PROGRAM P5_02_DiagramVisualisation
VAR
END_VAR
VAR // added by the converter: edge detectors and wires of the graphical bodies
    _w1, _w2, _w3 : BOOL;
    _w4 : INT;
END_VAR

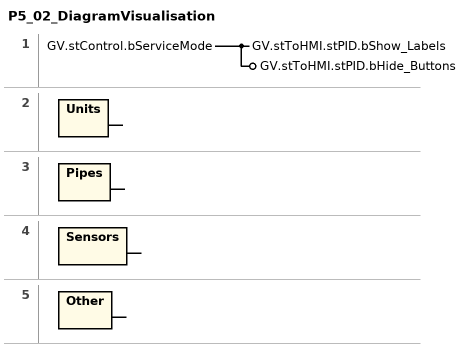
// NETWORK 1
_w1 := GV.stControl.bServiceMode;
GV.stToHMI.stPID.bShow_Labels := _w1;
GV.stToHMI.stPID.bHide_Buttons := NOT _w1;

// NETWORK 2
Units();

// NETWORK 3
Pipes();

// NETWORK 4
Sensors();

// NETWORK 5
Other();

ACTION Other:
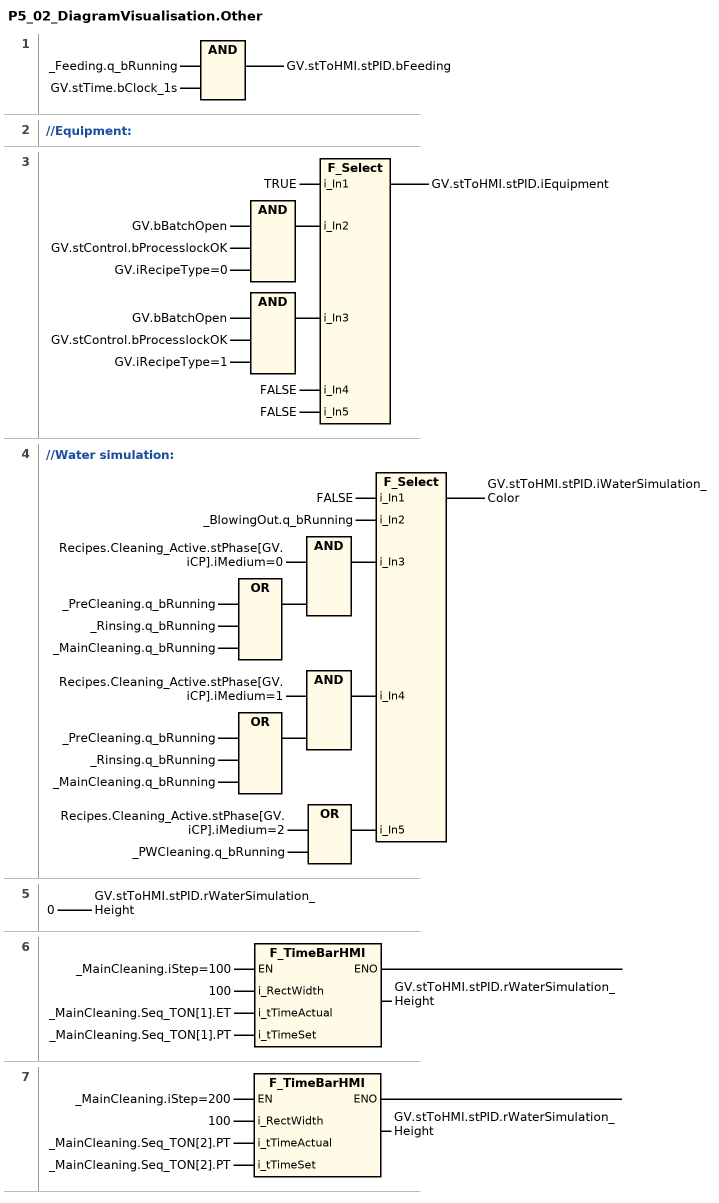
// NETWORK 1
GV.stToHMI.stPID.bFeeding := _Feeding.q_bRunning AND GV.stTime.bClock_1s;

// NETWORK 2
// label: //Equipment

// NETWORK 3
GV.stToHMI.stPID.iEquipment := F_Select(i_In1 := TRUE, i_In2 := GV.bBatchOpen AND GV.stControl.bProcesslockOK AND (GV.iRecipeType=0), i_In3 := GV.bBatchOpen AND GV.stControl.bProcesslockOK AND (GV.iRecipeType=1), i_In4 := FALSE, i_In5 := FALSE);

// NETWORK 4
// label: //Water simulation
GV.stToHMI.stPID.iWaterSimulation_Color := F_Select(i_In1 := FALSE, i_In2 := _BlowingOut.q_bRunning, i_In3 := (Recipes.Cleaning_Active.stPhase[GV.iCP].iMedium=0) AND (_PreCleaning.q_bRunning OR _Rinsing.q_bRunning OR _MainCleaning.q_bRunning), i_In4 := (Recipes.Cleaning_Active.stPhase[GV.iCP].iMedium=1) AND (_PreCleaning.q_bRunning OR _Rinsing.q_bRunning OR _MainCleaning.q_bRunning), i_In5 := (Recipes.Cleaning_Active.stPhase[GV.iCP].iMedium=2) OR _PWCleaning.q_bRunning);

// NETWORK 5
GV.stToHMI.stPID.rWaterSimulation_Height := 0;

// NETWORK 6
IF _MainCleaning.iStep=100 THEN
    GV.stToHMI.stPID.rWaterSimulation_Height := F_TimeBarHMI(i_RectWidth := 100, i_tTimeActual := _MainCleaning.Seq_TON[1].ET, i_tTimeSet := _MainCleaning.Seq_TON[1].PT);
END_IF

// NETWORK 7
IF _MainCleaning.iStep=200 THEN
    GV.stToHMI.stPID.rWaterSimulation_Height := F_TimeBarHMI(i_RectWidth := 100, i_tTimeActual := _MainCleaning.Seq_TON[2].PT, i_tTimeSet := _MainCleaning.Seq_TON[2].PT);
END_IF

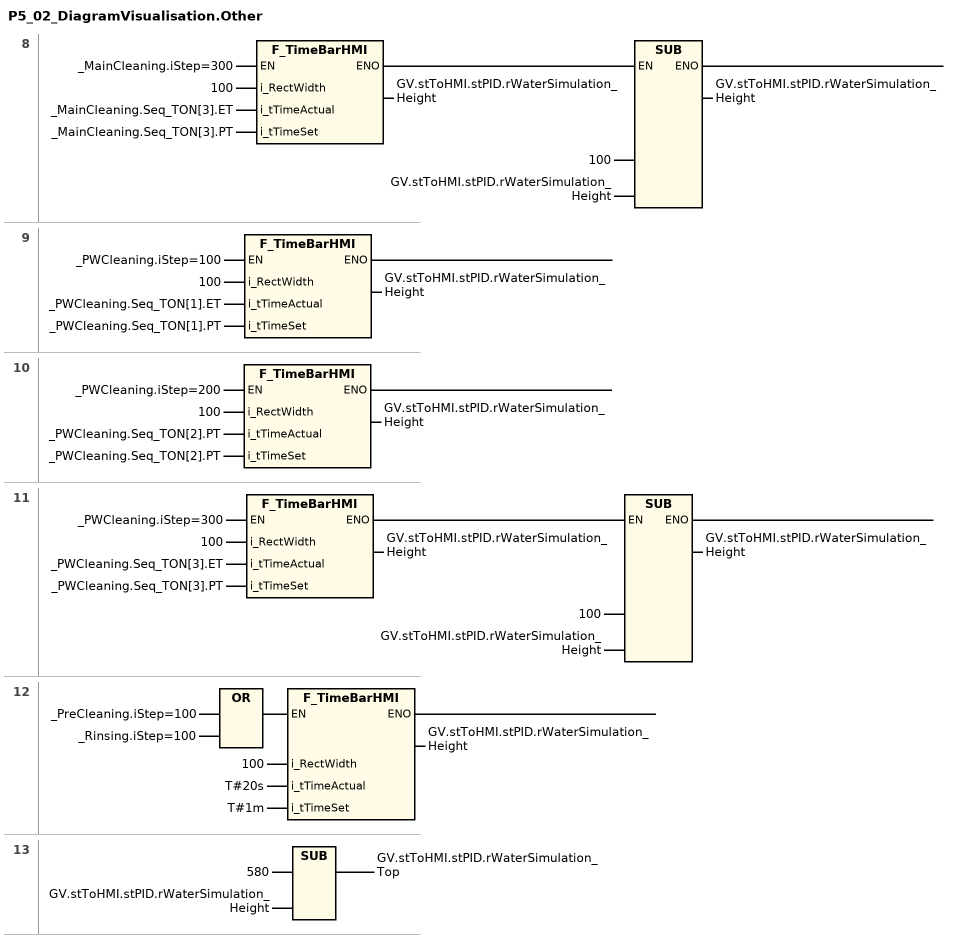
// NETWORK 8
_w2 := _MainCleaning.iStep=300;
IF _w2 THEN
    GV.stToHMI.stPID.rWaterSimulation_Height := F_TimeBarHMI(i_RectWidth := 100, i_tTimeActual := _MainCleaning.Seq_TON[3].ET, i_tTimeSet := _MainCleaning.Seq_TON[3].PT);
END_IF
IF _w2 THEN GV.stToHMI.stPID.rWaterSimulation_Height := 100 - GV.stToHMI.stPID.rWaterSimulation_Height; END_IF

// NETWORK 9
IF _PWCleaning.iStep=100 THEN
    GV.stToHMI.stPID.rWaterSimulation_Height := F_TimeBarHMI(i_RectWidth := 100, i_tTimeActual := _PWCleaning.Seq_TON[1].ET, i_tTimeSet := _PWCleaning.Seq_TON[1].PT);
END_IF

// NETWORK 10
IF _PWCleaning.iStep=200 THEN
    GV.stToHMI.stPID.rWaterSimulation_Height := F_TimeBarHMI(i_RectWidth := 100, i_tTimeActual := _PWCleaning.Seq_TON[2].PT, i_tTimeSet := _PWCleaning.Seq_TON[2].PT);
END_IF

// NETWORK 11
_w3 := _PWCleaning.iStep=300;
IF _w3 THEN
    GV.stToHMI.stPID.rWaterSimulation_Height := F_TimeBarHMI(i_RectWidth := 100, i_tTimeActual := _PWCleaning.Seq_TON[3].ET, i_tTimeSet := _PWCleaning.Seq_TON[3].PT);
END_IF
IF _w3 THEN GV.stToHMI.stPID.rWaterSimulation_Height := 100 - GV.stToHMI.stPID.rWaterSimulation_Height; END_IF

// NETWORK 12
IF (_PreCleaning.iStep=100) OR (_Rinsing.iStep=100) THEN
    GV.stToHMI.stPID.rWaterSimulation_Height := F_TimeBarHMI(i_RectWidth := 100, i_tTimeActual := T#20s, i_tTimeSet := T#1m);
END_IF

// NETWORK 13
GV.stToHMI.stPID.rWaterSimulation_Top := 580 - GV.stToHMI.stPID.rWaterSimulation_Height;
END_ACTION

ACTION Pipes:
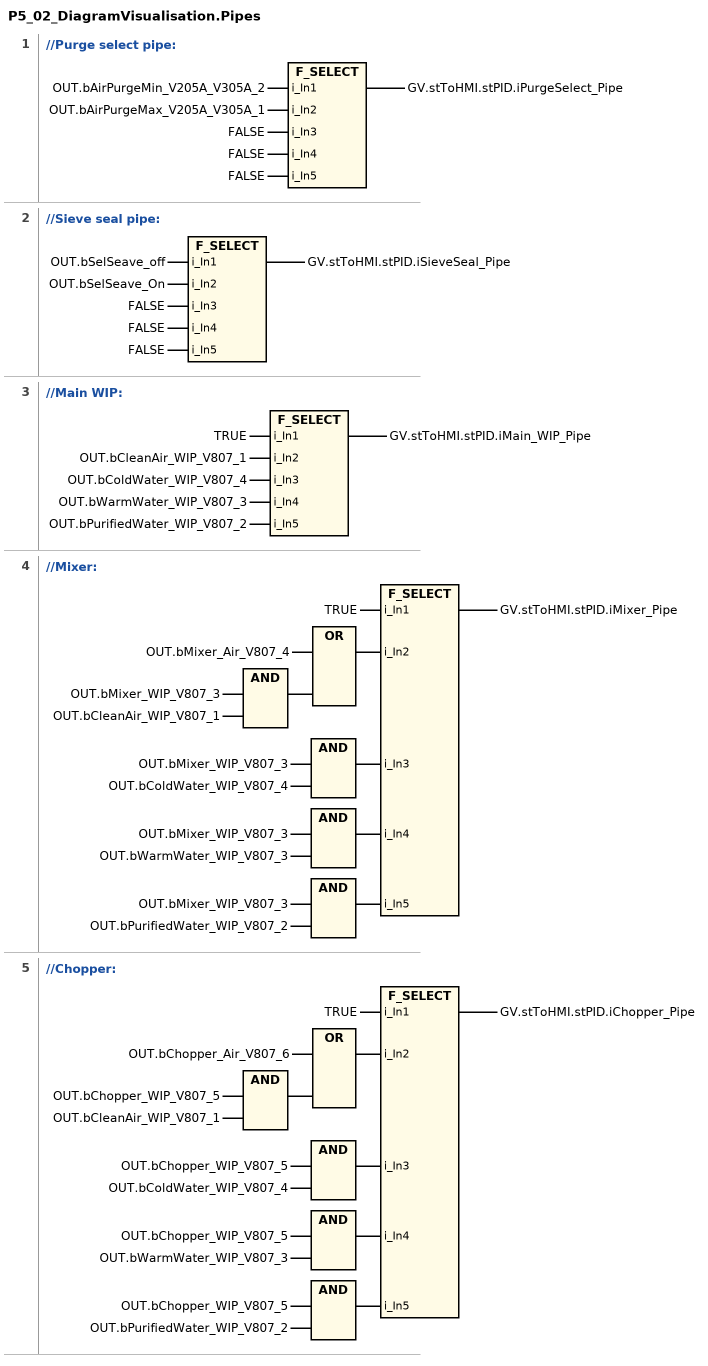
// NETWORK 1
// label: //Purge select pipe
GV.stToHMI.stPID.iPurgeSelect_Pipe := F_SELECT(i_In1 := OUT.bAirPurgeMin_V205A_V305A_2, i_In2 := OUT.bAirPurgeMax_V205A_V305A_1, i_In3 := FALSE, i_In4 := FALSE, i_In5 := FALSE);

// NETWORK 2
// label: //Sieve seal pipe
GV.stToHMI.stPID.iSieveSeal_Pipe := F_SELECT(i_In1 := OUT.bSelSeave_off, i_In2 := OUT.bSelSeave_On, i_In3 := FALSE, i_In4 := FALSE, i_In5 := FALSE);

// NETWORK 3
// label: //Main WIP
GV.stToHMI.stPID.iMain_WIP_Pipe := F_SELECT(i_In1 := TRUE, i_In2 := OUT.bCleanAir_WIP_V807_1, i_In3 := OUT.bColdWater_WIP_V807_4, i_In4 := OUT.bWarmWater_WIP_V807_3, i_In5 := OUT.bPurifiedWater_WIP_V807_2);

// NETWORK 4
// label: //Mixer
GV.stToHMI.stPID.iMixer_Pipe := F_SELECT(i_In1 := TRUE, i_In2 := OUT.bMixer_Air_V807_4 OR OUT.bMixer_WIP_V807_3 AND OUT.bCleanAir_WIP_V807_1, i_In3 := OUT.bMixer_WIP_V807_3 AND OUT.bColdWater_WIP_V807_4, i_In4 := OUT.bMixer_WIP_V807_3 AND OUT.bWarmWater_WIP_V807_3, i_In5 := OUT.bMixer_WIP_V807_3 AND OUT.bPurifiedWater_WIP_V807_2);

// NETWORK 5
// label: //Chopper
GV.stToHMI.stPID.iChopper_Pipe := F_SELECT(i_In1 := TRUE, i_In2 := OUT.bChopper_Air_V807_6 OR OUT.bChopper_WIP_V807_5 AND OUT.bCleanAir_WIP_V807_1, i_In3 := OUT.bChopper_WIP_V807_5 AND OUT.bColdWater_WIP_V807_4, i_In4 := OUT.bChopper_WIP_V807_5 AND OUT.bWarmWater_WIP_V807_3, i_In5 := OUT.bChopper_WIP_V807_5 AND OUT.bPurifiedWater_WIP_V807_2);

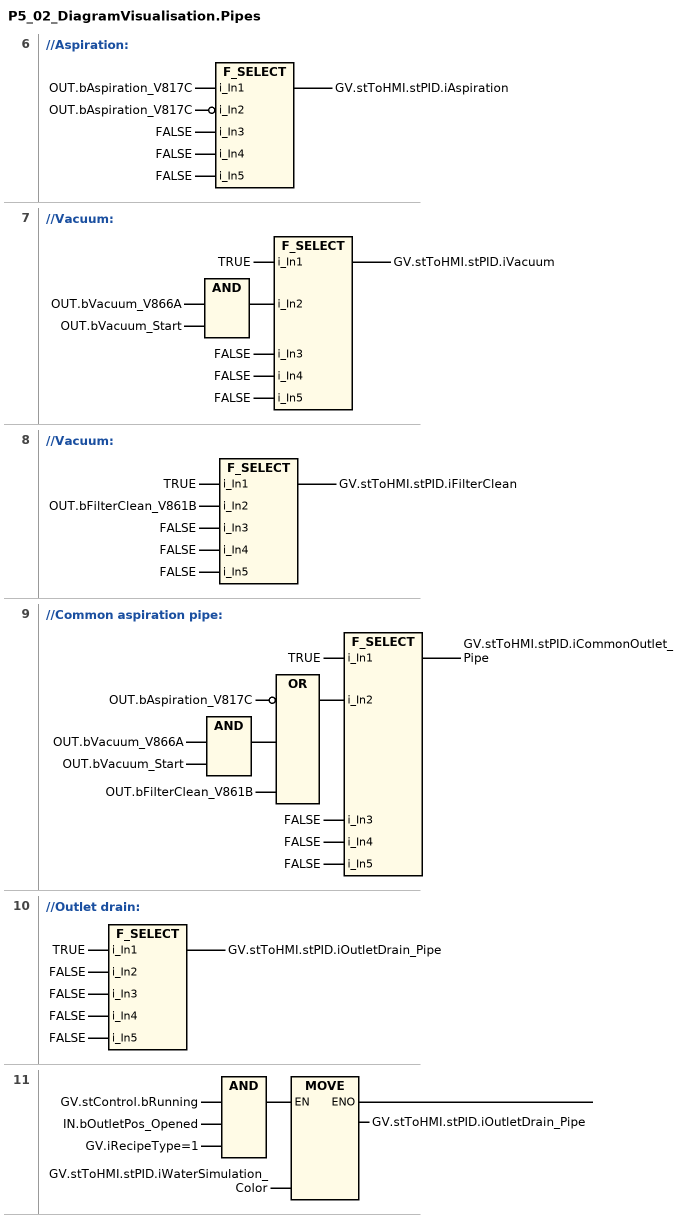
// NETWORK 6
// label: //Aspiration
GV.stToHMI.stPID.iAspiration := F_SELECT(i_In1 := OUT.bAspiration_V817C, i_In2 := NOT OUT.bAspiration_V817C, i_In3 := FALSE, i_In4 := FALSE, i_In5 := FALSE);

// NETWORK 7
// label: //Vacuum
GV.stToHMI.stPID.iVacuum := F_SELECT(i_In1 := TRUE, i_In2 := OUT.bVacuum_V866A AND OUT.bVacuum_Start, i_In3 := FALSE, i_In4 := FALSE, i_In5 := FALSE);

// NETWORK 8
// label: //Vacuum
GV.stToHMI.stPID.iFilterClean := F_SELECT(i_In1 := TRUE, i_In2 := OUT.bFilterClean_V861B, i_In3 := FALSE, i_In4 := FALSE, i_In5 := FALSE);

// NETWORK 9
// label: //Common aspiration pipe
GV.stToHMI.stPID.iCommonOutlet_Pipe := F_SELECT(i_In1 := TRUE, i_In2 := NOT OUT.bAspiration_V817C OR OUT.bVacuum_V866A AND OUT.bVacuum_Start OR OUT.bFilterClean_V861B, i_In3 := FALSE, i_In4 := FALSE, i_In5 := FALSE);

// NETWORK 10
// label: //Outlet drain
GV.stToHMI.stPID.iOutletDrain_Pipe := F_SELECT(i_In1 := TRUE, i_In2 := FALSE, i_In3 := FALSE, i_In4 := FALSE, i_In5 := FALSE);

// NETWORK 11
IF GV.stControl.bRunning AND IN.bOutletPos_Opened AND (GV.iRecipeType=1) THEN
    GV.stToHMI.stPID.iOutletDrain_Pipe := GV.stToHMI.stPID.iWaterSimulation_Color;
END_IF

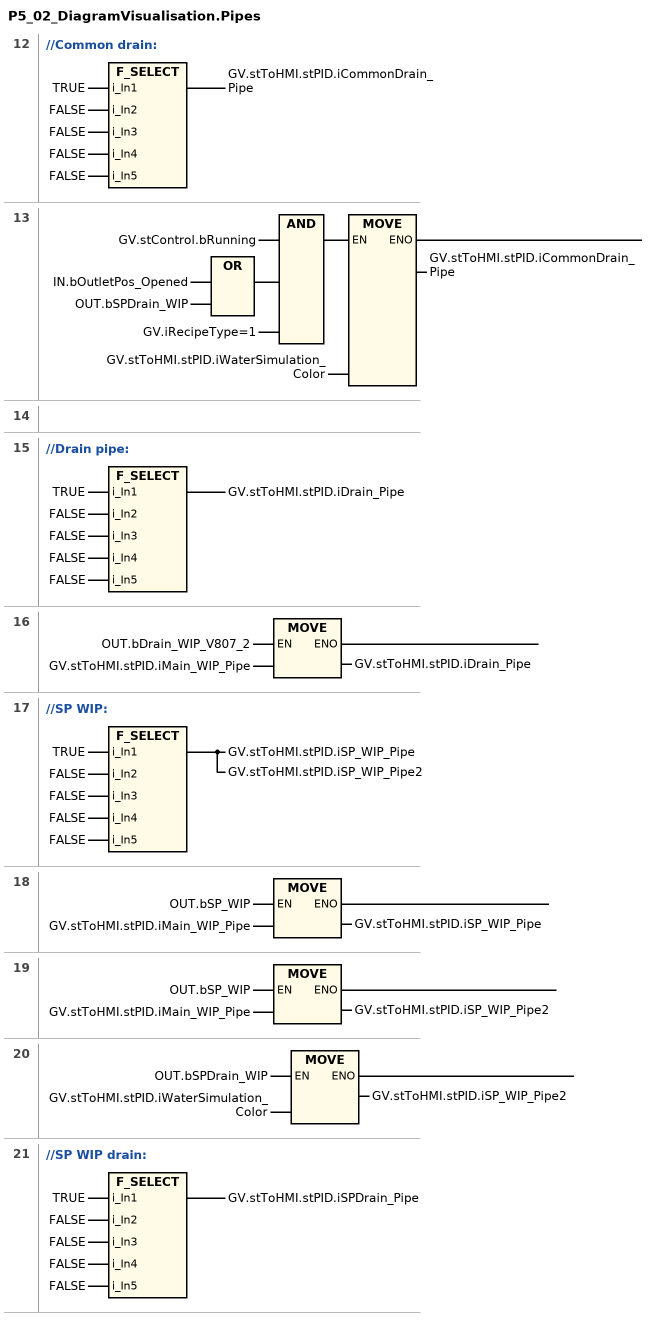
// NETWORK 12
// label: //Common drain
GV.stToHMI.stPID.iCommonDrain_Pipe := F_SELECT(i_In1 := TRUE, i_In2 := FALSE, i_In3 := FALSE, i_In4 := FALSE, i_In5 := FALSE);

// NETWORK 13
IF GV.stControl.bRunning AND (IN.bOutletPos_Opened OR OUT.bSPDrain_WIP) AND (GV.iRecipeType=1) THEN
    GV.stToHMI.stPID.iCommonDrain_Pipe := GV.stToHMI.stPID.iWaterSimulation_Color;
END_IF

// NETWORK 14

// NETWORK 15
// label: //Drain pipe
GV.stToHMI.stPID.iDrain_Pipe := F_SELECT(i_In1 := TRUE, i_In2 := FALSE, i_In3 := FALSE, i_In4 := FALSE, i_In5 := FALSE);

// NETWORK 16
IF OUT.bDrain_WIP_V807_2 THEN GV.stToHMI.stPID.iDrain_Pipe := GV.stToHMI.stPID.iMain_WIP_Pipe; END_IF

// NETWORK 17
// label: //SP WIP
_w4 := F_SELECT(i_In1 := TRUE, i_In2 := FALSE, i_In3 := FALSE, i_In4 := FALSE, i_In5 := FALSE);
GV.stToHMI.stPID.iSP_WIP_Pipe := _w4;
GV.stToHMI.stPID.iSP_WIP_Pipe2 := _w4;

// NETWORK 18
IF OUT.bSP_WIP THEN GV.stToHMI.stPID.iSP_WIP_Pipe := GV.stToHMI.stPID.iMain_WIP_Pipe; END_IF

// NETWORK 19
IF OUT.bSP_WIP THEN GV.stToHMI.stPID.iSP_WIP_Pipe2 := GV.stToHMI.stPID.iMain_WIP_Pipe; END_IF

// NETWORK 20
IF OUT.bSPDrain_WIP THEN GV.stToHMI.stPID.iSP_WIP_Pipe2 := GV.stToHMI.stPID.iWaterSimulation_Color; END_IF

// NETWORK 21
// label: //SP WIP drain
GV.stToHMI.stPID.iSPDrain_Pipe := F_SELECT(i_In1 := TRUE, i_In2 := FALSE, i_In3 := FALSE, i_In4 := FALSE, i_In5 := FALSE);

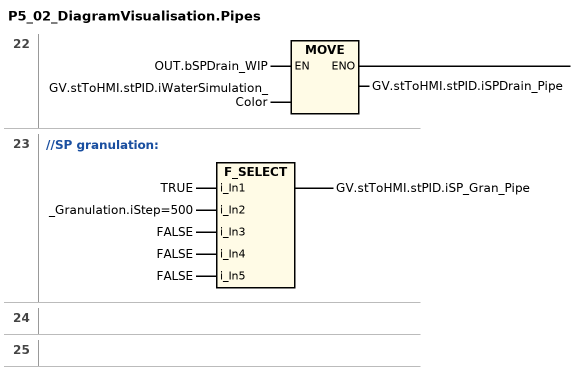
// NETWORK 22
IF OUT.bSPDrain_WIP THEN GV.stToHMI.stPID.iSPDrain_Pipe := GV.stToHMI.stPID.iWaterSimulation_Color; END_IF

// NETWORK 23
// label: //SP granulation
GV.stToHMI.stPID.iSP_Gran_Pipe := F_SELECT(i_In1 := TRUE, i_In2 := _Granulation.iStep=500, i_In3 := FALSE, i_In4 := FALSE, i_In5 := FALSE);

// NETWORK 24

// NETWORK 25
END_ACTION

ACTION Sensors:
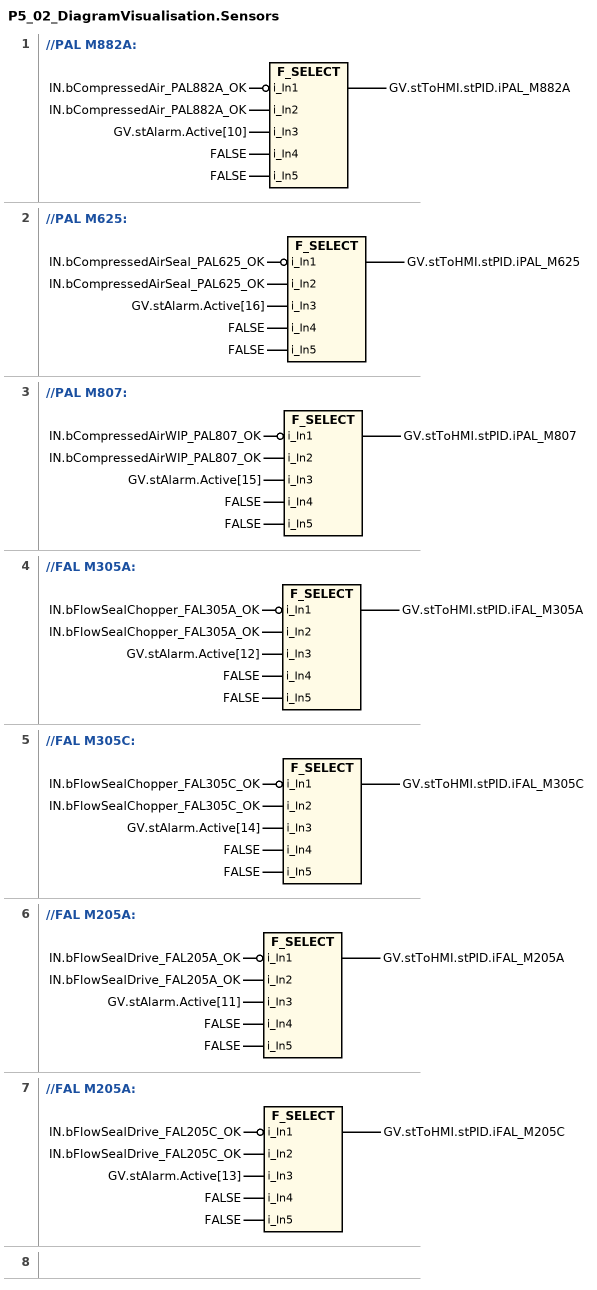
// NETWORK 1
// label: //PAL M882A
GV.stToHMI.stPID.iPAL_M882A := F_SELECT(i_In1 := NOT IN.bCompressedAir_PAL882A_OK, i_In2 := IN.bCompressedAir_PAL882A_OK, i_In3 := GV.stAlarm.Active[10], i_In4 := FALSE, i_In5 := FALSE);

// NETWORK 2
// label: //PAL M625
GV.stToHMI.stPID.iPAL_M625 := F_SELECT(i_In1 := NOT IN.bCompressedAirSeal_PAL625_OK, i_In2 := IN.bCompressedAirSeal_PAL625_OK, i_In3 := GV.stAlarm.Active[16], i_In4 := FALSE, i_In5 := FALSE);

// NETWORK 3
// label: //PAL M807
GV.stToHMI.stPID.iPAL_M807 := F_SELECT(i_In1 := NOT IN.bCompressedAirWIP_PAL807_OK, i_In2 := IN.bCompressedAirWIP_PAL807_OK, i_In3 := GV.stAlarm.Active[15], i_In4 := FALSE, i_In5 := FALSE);

// NETWORK 4
// label: //FAL M305A
GV.stToHMI.stPID.iFAL_M305A := F_SELECT(i_In1 := NOT IN.bFlowSealChopper_FAL305A_OK, i_In2 := IN.bFlowSealChopper_FAL305A_OK, i_In3 := GV.stAlarm.Active[12], i_In4 := FALSE, i_In5 := FALSE);

// NETWORK 5
// label: //FAL M305C
GV.stToHMI.stPID.iFAL_M305C := F_SELECT(i_In1 := NOT IN.bFlowSealChopper_FAL305C_OK, i_In2 := IN.bFlowSealChopper_FAL305C_OK, i_In3 := GV.stAlarm.Active[14], i_In4 := FALSE, i_In5 := FALSE);

// NETWORK 6
// label: //FAL M205A
GV.stToHMI.stPID.iFAL_M205A := F_SELECT(i_In1 := NOT IN.bFlowSealDrive_FAL205A_OK, i_In2 := IN.bFlowSealDrive_FAL205A_OK, i_In3 := GV.stAlarm.Active[11], i_In4 := FALSE, i_In5 := FALSE);

// NETWORK 7
// label: //FAL M205A
GV.stToHMI.stPID.iFAL_M205C := F_SELECT(i_In1 := NOT IN.bFlowSealDrive_FAL205C_OK, i_In2 := IN.bFlowSealDrive_FAL205C_OK, i_In3 := GV.stAlarm.Active[13], i_In4 := FALSE, i_In5 := FALSE);

// NETWORK 8
END_ACTION

ACTION Units:
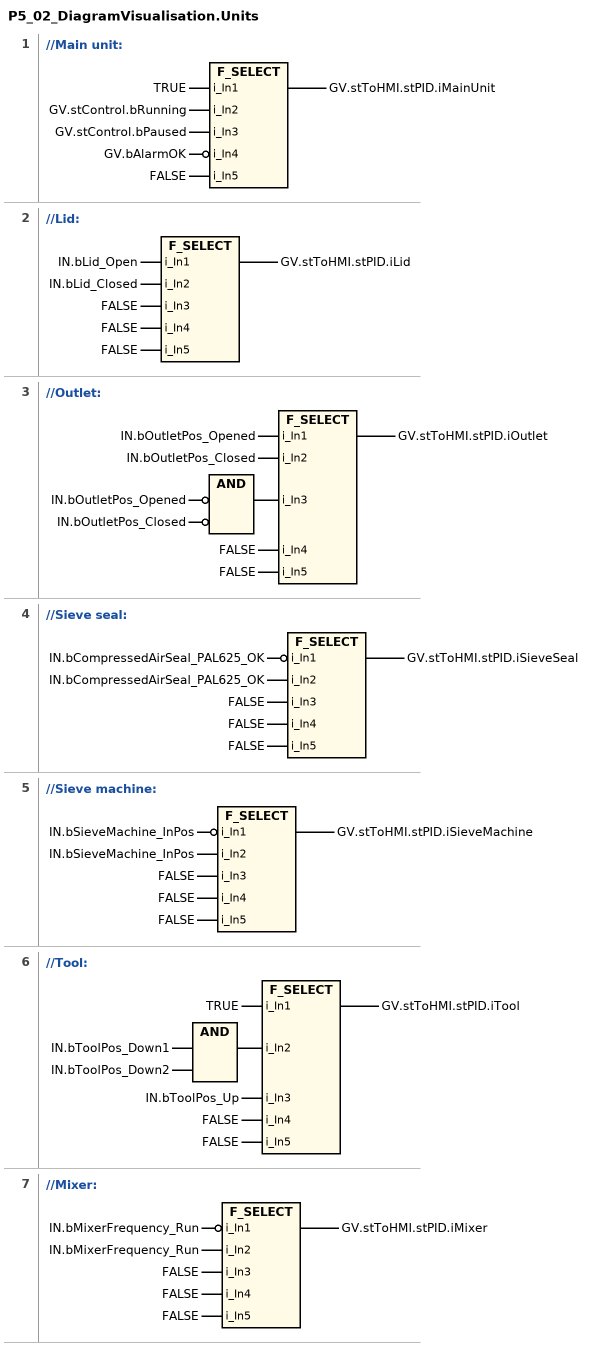
// NETWORK 1
// label: //Main unit
GV.stToHMI.stPID.iMainUnit := F_SELECT(i_In1 := TRUE, i_In2 := GV.stControl.bRunning, i_In3 := GV.stControl.bPaused, i_In4 := NOT GV.bAlarmOK, i_In5 := FALSE);

// NETWORK 2
// label: //Lid
GV.stToHMI.stPID.iLid := F_SELECT(i_In1 := IN.bLid_Open, i_In2 := IN.bLid_Closed, i_In3 := FALSE, i_In4 := FALSE, i_In5 := FALSE);

// NETWORK 3
// label: //Outlet
GV.stToHMI.stPID.iOutlet := F_SELECT(i_In1 := IN.bOutletPos_Opened, i_In2 := IN.bOutletPos_Closed, i_In3 := NOT IN.bOutletPos_Opened AND NOT IN.bOutletPos_Closed, i_In4 := FALSE, i_In5 := FALSE);

// NETWORK 4
// label: //Sieve seal
GV.stToHMI.stPID.iSieveSeal := F_SELECT(i_In1 := NOT IN.bCompressedAirSeal_PAL625_OK, i_In2 := IN.bCompressedAirSeal_PAL625_OK, i_In3 := FALSE, i_In4 := FALSE, i_In5 := FALSE);

// NETWORK 5
// label: //Sieve machine
GV.stToHMI.stPID.iSieveMachine := F_SELECT(i_In1 := NOT IN.bSieveMachine_InPos, i_In2 := IN.bSieveMachine_InPos, i_In3 := FALSE, i_In4 := FALSE, i_In5 := FALSE);

// NETWORK 6
// label: //Tool
GV.stToHMI.stPID.iTool := F_SELECT(i_In1 := TRUE, i_In2 := IN.bToolPos_Down1 AND IN.bToolPos_Down2, i_In3 := IN.bToolPos_Up, i_In4 := FALSE, i_In5 := FALSE);

// NETWORK 7
// label: //Mixer
GV.stToHMI.stPID.iMixer := F_SELECT(i_In1 := NOT IN.bMixerFrequency_Run, i_In2 := IN.bMixerFrequency_Run, i_In3 := FALSE, i_In4 := FALSE, i_In5 := FALSE);

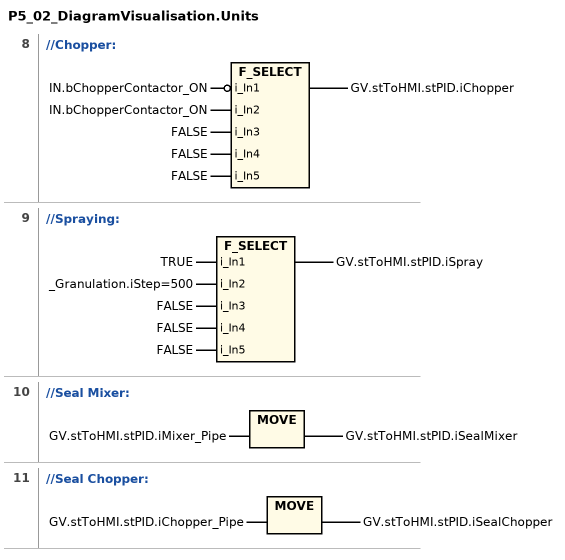
// NETWORK 8
// label: //Chopper
GV.stToHMI.stPID.iChopper := F_SELECT(i_In1 := NOT IN.bChopperContactor_ON, i_In2 := IN.bChopperContactor_ON, i_In3 := FALSE, i_In4 := FALSE, i_In5 := FALSE);

// NETWORK 9
// label: //Spraying
GV.stToHMI.stPID.iSpray := F_SELECT(i_In1 := TRUE, i_In2 := _Granulation.iStep=500, i_In3 := FALSE, i_In4 := FALSE, i_In5 := FALSE);

// NETWORK 10
// label: //Seal Mixer
GV.stToHMI.stPID.iSealMixer := GV.stToHMI.stPID.iMixer_Pipe;

// NETWORK 11
// label: //Seal Chopper
GV.stToHMI.stPID.iSealChopper := GV.stToHMI.stPID.iChopper_Pipe;
END_ACTION

END_PROGRAM

(* stored: Version 1.1.0.1, ProductVersion 3.1.4026.13
   POU P5_02_DiagramVisualisation: Id {bc9e8a74-853f-4307-bdae-27c231815e17}, SpecialFunc None
   Action Other: Id {5626b749-3c68-4497-b56e-ed4eebdc851d}
   Action Pipes: Id {245dfbe3-a9a8-456b-879f-74ca82b0a057}
   Action Sensors: Id {18a46ace-4f7d-4139-9dca-cf81f35cf47b}
   Action Units: Id {d1ca0c0c-5666-403c-8118-50fa95a64fcc} *)
